ORGANIZATION_BLOCK MAIN:OB1
TITLE=
BEGIN
Network 1 // �״�ɨ���ʼ��
LD     SM0.1
MOVB   0, VB100
MOVB   0, VB101
R      Q0.0, 8
R      Q1.0, 1
R      M0.0, 2
MOVW   13824, VW1120
MOVW   13824, VW1122

Network 2 // ÿɨ�豣��HSC����
LD     SM0.0
MOVB   16#F8, SMB37
MOVD   +0, SMD38
MOVD   +2000000000, SMD42
HDEF   0, 0
HSC    0
MOVB   16#F8, SMB47
MOVD   +0, SMD48
MOVD   +2000000000, SMD52
HDEF   1, 0
HSC    1

Network 3 // ��ͣ����
LD     I0.3
MOVB   0, VB100
MOVB   0, VB101
R      Q0.0, 8
R      Q1.0, 1
R      M0.0, 2
MOVW   13824, VW1120
MOVW   13824, VW1122

Network 4 // ��������
LD     I0.1
AN     I0.3
AB=    VB100, 0
AB=    VB101, 0
MOVB   10, VB100

Network 5 // �ػ�����
LD     I0.2
AN     I0.3
MOVB   0, VB100
MOVB   10, VB101

Network 6 // AE08ѹ��
LD     SM0.0
MOVW   AIW16, VW1000

Network 7 // AE08����Һλ
LD     SM0.0
MOVW   AIW18, VW1002

Network 8 // AE08����Һλ
LD     SM0.0
MOVW   AIW20, VW1004

Network 9 // ��������10
LD     SM0.0
AB=    VB100, 10
S      Q0.7, 1
S      Q0.2, 1
S      Q0.3, 1

Network 10 // ��������10�������
LD     SM0.0
AB=    VB100, 10
AW>=   VW1002, 100
R      Q0.2, 1

Network 11 // ��������10�������
LD     SM0.0
AB=    VB100, 10
AW>=   VW1004, 100
R      Q0.3, 1

Network 12 // ��������10ת20
LD     SM0.0
AB=    VB100, 10
AN     Q0.2
AN     Q0.3
MOVB   20, VB100

Network 13 // ��������20
LD     SM0.0
AB=    VB100, 20
S      Q0.6, 1
TON    T37, 30

Network 14 // ��������20ת30
LD     SM0.0
AB=    VB100, 20
A      T37
MOVB   30, VB100

Network 15 // ��������30
LD     SM0.0
AB=    VB100, 30
S      Q0.4, 1
TON    T38, 30

Network 16 // ��������30ת40
LD     SM0.0
AB=    VB100, 30
A      T38
MOVB   40, VB100

Network 17 // ��������40
LD     SM0.0
AB=    VB100, 40
S      M0.0, 1

Network 18 // ��������40ת50
LD     SM0.0
AB=    VB100, 40
AW>=   VW1000, 1000
MOVB   50, VB100

Network 19 // ��������50
LD     SM0.0
AB=    VB100, 50
S      M0.1, 1
TON    T39, 30

Network 20 // ��������50ת60
LD     SM0.0
AB=    VB100, 50
A      T39
MOVB   60, VB100

Network 21 // ��������60
LD     SM0.0
AB=    VB100, 60
S      Q0.5, 1
TON    T40, 3000

Network 22 // ��������60ת70
LD     SM0.0
AB=    VB100, 60
A      T40
MOVB   70, VB100

Network 23 // ��������70
LD     SM0.0
AB=    VB100, 70
S      Q1.0, 1
MOVB   100, VB100

Network 24 // �ػ�����10
LD     SM0.0
AB=    VB101, 10
R      Q1.0, 1
R      Q0.2, 2
R      Q0.7, 1
R      M0.1, 1
R      Q0.5, 1
R      M0.0, 1
R      Q0.4, 1
MOVB   20, VB101

Network 25 // �ػ�����20
LD     SM0.0
AB=    VB101, 20
TON    T41, 18000

Network 26 // AQ02����ʹ��
LD     M0.0
MOVW   VW1120, AQW32

Network 27 // AQ02����δʹ��
LD     SM0.0
AN     M0.0
MOVW   0, AQW32

Network 28 // AQ02����ʹ��
LD     M0.1
MOVW   VW1122, AQW34

Network 29 // AQ02����δʹ��
LD     SM0.0
AN     M0.1
MOVW   0, AQW34

Network 30 // 1����ٽ�����
LD     SM0.0
AN     M10.0
TON    T42, +10

Network 31 // ������1����
LD     T42
S      M10.0, 1
MOVD   HC0, VD1200
MOVD   VD1200, VD1208
-D     VD1204, VD1208
MOVD   VD1200, VD1204

Network 32 // ������2����
LD     T42
MOVD   HC1, VD1220
MOVD   VD1220, VD1228
-D     VD1224, VD1228
MOVD   VD1220, VD1224

Network 33 // ���ĸ�λ
LD     M10.0
AN     T42
R      M10.0, 1

Network 34 // ������1����ת
LD     SM0.0
DTR    VD1208, VD1300
DTR    VD1200, VD1304

Network 35 // ������1˲ʱ����
LD     SM0.0
MOVR   VD1300, VD1310
*R     60.0, VD1310
/R     2223.0, VD1310

Network 36 // ������1�ۼ�����
LD     SM0.0
MOVR   VD1304, VD1314
/R     2223.0, VD1314

Network 37 // ������2����ת
LD     SM0.0
DTR    VD1228, VD1320
DTR    VD1220, VD1324

Network 38 // ������2˲ʱ����
LD     SM0.0
MOVR   VD1320, VD1330
*R     60.0, VD1330
/R     2223.0, VD1330

Network 39 // ������2�ۼ�����
LD     SM0.0
MOVR   VD1324, VD1334
/R     2223.0, VD1334

END_ORGANIZATION_BLOCK
